FUNCTION_BLOCK Init
VAR_INPUT
END_VAR
VAR_OUTPUT
END_VAR
VAR
	isInit: BOOL := FALSE;
END_VAR

IF NOT isInit AND GVL.ToggleSwitch = FALSE THEN
	IF NOT GVL.KSV THEN
		AUTO.MotorIzbira := 1;
		AUTO.VrtenjeSmer := TRUE;
		AUTO.VrtenjePremik := TRUE;
	ELSIF NOT GVL.KSD THEN
		AUTO.VrtenjePremik:= FALSE;
		AUTO.MotorIzbira := 2;
		AUTO.DvigSmer := TRUE;
		AUTO.DvigPremik := TRUE;
	ELSIF NOT GVL.KSP THEN
		AUTO.MotorIzbira := 4;
		AUTO.PrijemSmer := TRUE;
		AUTO.PrijemPremik := TRUE;
	ELSE
		AUTO.MotorIzbira := 0;
		AUTO.Current.Y := 0;
		IF GVL.ULBButton = TRUE THEN
			AUTO.Recept := 1;
		ELSIF GVL.URBButton = TRUE THEN
			AUTO.Recept:= 2;
		ELSIF GVL.LLBButton= TRUE THEN
			AUTO.Recept := 3;
		END_IF
		IF AUTO.Recept <> 0 THEN
			AUTO.StageSelect := 1;
			isInit := TRUE;
		END_IF
		
	END_IF
END_IF

END_FUNCTION_BLOCK

(* stored: Version 1.1.0.1, ProductVersion 3.1.4024.12
   POU Init: Id {58081b1d-844a-491d-9e19-8082773cf0bf}, SpecialFunc None *)
